SYSTEM test
  (* Version 1.0, 2025-01-31, franz *)
  APPLICATION App
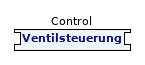
    SUBAPPS
      Control : Ventilsteuerung;
    END_SUBAPPS
  END_APPLICATION
  DEVICE FORTE_PC : FORTE_PC(MGR_ID := C_ST (* Device manager socket ID *))
    {SET_ATTRIBUTE(Profile, HOLOBLOC)}
    RESOURCE EMB_RES : EMB_RES
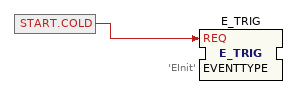
      FBS
        E_TRIG : E_TRIG(EVENTTYPE := 'EInit');
      END_FBS
      EVENT_CONNECTIONS
        START.COLD TO E_TRIG.REQ;
      END_CONNECTIONS
    END_RESOURCE
  END_DEVICE
  MAPPINGS
    App.Control ON FORTE_PC.EMB_RES;
  END_MAPPINGS
  SEGMENTS
    Ethernet : Ethernet;
  END_SEGMENTS
  LINKS
    FORTE_PC => Ethernet;
  END_LINKS
END_SYSTEM
